FUNCTION SetVec3 : Vec3
VAR_INPUT
	a,b,c : LREAL;
END_VAR
VAR
END_VAR

SetVec3.data[0] := a;
SetVec3.data[1] := b;
SetVec3.data[2] := c;

END_FUNCTION

(* stored: Version 1.1.0.1, ProductVersion 3.1.4024.2
   POU SetVec3: Id {68a40bf6-8eb8-42ec-bb2a-85ae7114286a}, SpecialFunc None *)
